Fanuc KAREL source: kb00030.KL

-- PROVISIONAL review KL for V1013-1; original PC SHA256 77106d24bf5c3d7cffda5c1090e87aed9cc1ba1d7047cb7050332eee435813f5
-- Incomplete behavior may be omitted. Consult companion uncertainty JSON. Do not deploy.
PROGRAM KB00030
%NOLOCKGROUP
BEGIN
  -- UNRESOLVED_PC offsets 5-12; opcodes 9D,23
  -- UNRESOLVED_PC offsets 17-24; opcodes 9D,23
  -- UNRESOLVED_PC offsets 29-38; opcodes 3F,75
  -- UNRESOLVED_PC offsets 43-50; opcodes 9D,23
  -- UNRESOLVED_PC offsets 55-85; opcodes 27,22,22,22,2A,22,31
  -- UNRESOLVED_PC offsets 90-94; opcodes 7F
END KB00030
